TYPE "UDT_MES_LoadData"
VERSION : 0.1
   STRUCT
      "PLC.PartTypeID" : Int;
      "PLC.PartSN" : String[50];
      "PLC.SubPartID" : String[50];
      "MES.ErrorCode" : Int;
      "MES.ErrorMsg" : String[50];
      "MES.StatusBits" : DInt;
      "MES.Cycle_ID" : DInt;
      "MES.Unit_ParttypeID" : Int;
   END_STRUCT;

END_TYPE

